FUNCTION F_Trend : BOOL
VAR_INPUT
	fCurrentValue	: REAL;
END_VAR
VAR_IN_OUT
	fValueMax		: REAL;
	fValueMin		: REAL;	
END_VAR

IF (fCurrentValue > fValueMax) THEN
	fValueMax:=fCurrentValue;
ELSIF (fCurrentValue < fValueMax) THEN
	fValueMin:= fCurrentValue;
END_IF

END_FUNCTION

(* stored: Version 1.1.0.1, ProductVersion 3.1.4024.11
   POU F_Trend: Id {cadcebf4-3c09-4d1b-9288-7604522ea0a8}, SpecialFunc None *)
